// this function is used to check if input statament is true.
// if false, the code will trigger a zero-devide exception and stop the whole program by PLC
FUNCTION ASSERT : BOOL
VAR_INPUT
	statement:BOOL;
END_VAR
VAR
	zero:INT :=0;
	res :REAL:=0;
END_VAR

IF NOT(statement) THEN
	res := 1/zero;
END_IF

ASSERT := true;

END_FUNCTION

(* stored: Version 1.1.0.1, ProductVersion 3.1.4024.12
   POU ASSERT: Id {ba49b7c8-3131-4df5-a3e8-52027de90f57}, SpecialFunc None *)
